(* IEC 61131-3 sources: PLC-programming-/, 3 files *)

(* ---- trial1.st ---- *)
PROGRAM program0
  VAR
    sensor AT %IX100.0 : BOOL;
    running AT %IX100.1 : BOOL;
    conveyor1 AT %QX100.0 : BOOL;
  END_VAR

  IF running = TRUE THEN
    conveyor1 := TRUE;
  ELSIF sensor = FALSE THEN
    conveyor1 := FALSE;
  END_IF;

END_PROGRAM

CONFIGURATION Config0

  RESOURCE Res0 ON PLC
    TASK task0(INTERVAL := T#20ms,PRIORITY := 0);
    PROGRAM instance0 WITH task0 : program0;
  END_RESOURCE
END_CONFIGURATION

(* ---- trial2.st ---- *)
PROGRAM program0
  VAR
    sensor AT %IX100.0 : BOOL;
    running AT %IX100.1 : BOOL;
    conveyor1 AT %QX100.0 : BOOL;
  END_VAR

  IF running = TRUE AND NOT sensor THEN
    conveyor1 := TRUE;
  ELSIF sensor = FALSE THEN
    conveyor1 := FALSE;
  END_IF;

END_PROGRAM

CONFIGURATION Config0

  RESOURCE Res0 ON PLC
    TASK task0(INTERVAL := T#20ms,PRIORITY := 0);
    PROGRAM instance0 WITH task0 : program0;
  END_RESOURCE
END_CONFIGURATION

(* ---- trial3.st ---- *)
PROGRAM program0
  VAR
    sensor AT %IX100.0 : BOOL;
    running AT %IX100.1 : BOOL;
    conveyor1 AT %QX100.0 : BOOL;
  END_VAR

  IF running = TRUE THEN
    conveyor1 := TRUE;
  END_IF;
  IF sensor = FALSE THEN
    conveyor1 := FALSE;
  END_IF;
END_PROGRAM

CONFIGURATION Config0

  RESOURCE Res0 ON PLC
    TASK task0(INTERVAL := T#20ms,PRIORITY := 0);
    PROGRAM instance0 WITH task0 : program0;
  END_RESOURCE
END_CONFIGURATION
